FUNCTION_BLOCK FB_INT_TO_BCD_WORD (* Convert INT to 4 BCD digits *)
  (* Standard: 61499-1; Classification: Simple FB; Function: BCD conversion; Type: INT to WORD *)
  (* Version 0.0, 2007-08-27, JHC, Holobloc Inc *)
  (* Compiler header: package fb.rt.math; *)
  (* Compiler classdef: SimpleFB *)
  (* Compiler Java Sun JDK 1.6.0 *)
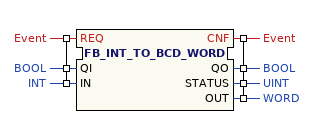
  EVENT_INPUT
    REQ WITH QI, IN; (* Normal Execution Request *)
  END_EVENT
  EVENT_OUTPUT
    CNF WITH QO, STATUS, OUT; (* Execution Confirmation *)
  END_EVENT
  VAR_INPUT
    QI : BOOL; (* Input event qualifier *)
    IN : INT; (* 0<=IN<=9999 *)
  END_VAR
  VAR_OUTPUT
    QO : BOOL; (* Output event qualifier *)
    STATUS : UINT; (* 0=OK, 2=conversion error per 61499-1 Table D.1 *)
    OUT : WORD; (* BCD value of IN *)
  END_VAR
  ALGORITHM REQ IN Java: (* Normally executed algorithm *)
QO.value=QI.value;
  END_ALGORITHM
END_FUNCTION_BLOCK
